PROGRAM prgSystemTime
VAR
	fbGetTime			: NT_GetTime;
	dtSystemTime		: DT;
	stDateTime			: TIMESTRUCT;
	tonGetTime			: TON;
	nStep				: INT;
	bSystemTimeValid	: BOOL := FALSE;
END_VAR

CASE nStep OF
0:
	tonGetTime(IN:=TRUE, PT:=T#500MS);
	IF (tonGetTime.Q) THEN
		tonGetTime(IN := FALSE);
		nStep:=10;
	END_IF

10:
	fbGetTime(NETID:='', START:=TRUE, TMOUT:=T#2S);
	IF (NOT fbGetTime.BUSY) THEN
		stDateTime := fbGetTime.TIMESTR;
		dtSystemTime := SYSTEMtimE_TO_DT(fbGetTime.TIMESTR);
		fbGetTime(START := FALSE);
		bSystemTimeValid := TRUE;
		nStep := 0;
	END_IF	
END_CASE

END_PROGRAM

(* stored: Version 1.1.0.1, ProductVersion 3.1.4024.9
   POU prgSystemTime: Id {ebee8292-6ded-45d7-be6e-5d3afc86b167}, SpecialFunc None *)
